    IF Error = 1 THEN 
        (* '<S2>:1:33' x = x0; *)
        PositionRef_m := fCylPos0_m;
        (* '<S2>:1:34' v = v0; *)
        VelocityRef_ms := fCylVel0_ms;
    ELSIF (fSimulationTime_s >= 0.0) AND (fSimulationTime_s < ft0_s) THEN 
        (* '<S2>:1:35' elseif t>=0 && t<t0 *)
        (* '<S2>:1:36' x = x0; *)
        PositionRef_m := fCylPos0_m;
        (* '<S2>:1:37' v = v0; *)
        VelocityRef_ms := fCylVel0_ms;
    ELSIF (fSimulationTime_s >= ft0_s) AND (fSimulationTime_s < x2_tmp_tmp) THEN 
        (* '<S2>:1:38' elseif t>=t0 && t<(t0+t1) *)
        (* '<S2>:1:39' x = x0 + v0*(t-t0)-(slopeExt/t1)*(t-t0)^2/2; *)
        slopeRetr := fSimulationTime_s - ft0_s;
        PositionRef_m := ((slopeRetr * fCylVel0_ms) + fCylPos0_m) - ((x1_tmp_tmp * (slopeRetr * slopeRetr)) / 2.0);
        (* '<S2>:1:40' v = v0-(slopeExt/t1)*(t-t0); *)
        VelocityRef_ms := fCylVel0_ms - (x1_tmp_tmp * slopeRetr);
    ELSIF (fSimulationTime_s >= x2_tmp_tmp) AND (fSimulationTime_s < x2_tmp) THEN 
        (* '<S2>:1:41' elseif t>=(t0+t1) && t<(t0+t1+t2) *)
        (* '<S2>:1:42' x = x1 + vs*(t-(t0+t1)); *)
        PositionRef_m := ((fSimulationTime_s - x2_tmp_tmp) * fVelocitySP_ms) + x1;
        (* '<S2>:1:43' v = vs; *)
        VelocityRef_ms := fVelocitySP_ms;
    ELSIF (fSimulationTime_s >= x2_tmp) AND (fSimulationTime_s < x4_tmp_tmp) THEN 
        (* '<S2>:1:44' elseif t>=(t0+t1+t2) && t<(t0+t1+t2+t3) *)
        (* '<S2>:1:45' x = x2+vs*(t-(t0+t1+t2))+(slopeExt/t3)*(t-(t0+t1+t2))^2/2; *)
        slopeRetr := fSimulationTime_s - ((ft0_s + ftRamp_s) + tHold);
        PositionRef_m := ((slopeRetr * fVelocitySP_ms) + x2) + ((x1_tmp_tmp * (slopeRetr * slopeRetr)) / 2.0);
        (* '<S2>:1:46' v = vs+(slopeExt/t3)*(t-(t0+t1+t2)); *)
        VelocityRef_ms := (slopeRetr * (slopeExt / ftRamp_s)) + fVelocitySP_ms;
    ELSIF (fSimulationTime_s >= x4_tmp_tmp) AND (fSimulationTime_s < x4_tmp) THEN 
        (* '<S2>:1:47' elseif t>=(t0+t1+t2+t3) && t<(t0+t1+t2+t3+t4) *)
        (* '<S2>:1:48' x = x_ref; *)
        PositionRef_m := fPositionSP_m;
        (* '<S2>:1:49' v = v0; *)
        VelocityRef_ms := fCylVel0_ms;
    ELSE 
        x1_tmp_tmp := ((x2_tmp_tmp + tHold) + ftRamp_s) + ftHoldPos_s;
        slopeExt := x1_tmp_tmp + ftRamp_s;

        IF (fSimulationTime_s >= x1_tmp_tmp) AND (fSimulationTime_s < slopeExt) THEN 
            (* '<S2>:1:50' elseif t>=(t0+t1+t2+t3+t4) && t<(t0+t1+t2+t3+t4+t5) *)
            (* '<S2>:1:51' x = x_ref - v0*(t-(t0+t1+t2+t3+t4))+(slopeRetr/t5)*(t-(t0+t1+t2+t3+t4))^2/2; *)
            tHold := fSimulationTime_s - x1_tmp_tmp;
            slopeRetr := slopeRetr / ftRamp_s;
            PositionRef_m := (fPositionSP_m - (tHold * fCylVel0_ms)) + ((slopeRetr * (tHold * tHold)) / 2.0);
            (* '<S2>:1:52' v = v0+(slopeRetr/t5)*(t-(t0+t1+t2+t3+t4)); *)
            VelocityRef_ms := (tHold * slopeRetr) + fCylVel0_ms;
        ELSE 
            x1_tmp_tmp := slopeExt + tHold;

            IF (fSimulationTime_s >= slopeExt) AND (fSimulationTime_s < x1_tmp_tmp) THEN 
                (* '<S2>:1:53' elseif t>=(t0+t1+t2+t3+t4+t5) && t<(t0+t1+t2+t3+t4+t5+t6) *)
                (* '<S2>:1:54' x = x4-vs*(t-(t0+t1+t2+t3+t4+t5)); *)
                PositionRef_m := x4 - ((fSimulationTime_s - slopeExt) * fVelocitySP_ms);
                (* '<S2>:1:55' v = -vs; *)
                VelocityRef_ms :=  -fVelocitySP_ms;
            ELSIF (fSimulationTime_s >= x1_tmp_tmp) AND (fSimulationTime_s < (x1_tmp_tmp + ftRamp_s)) THEN 
                (* '<S2>:1:56' elseif t>=(t0+t1+t2+t3+t4+t5+t6) && t<(t0+t1+t2+t3+t4+t5+t6+t7) *)
                (* '<S2>:1:57' x = x5-vs*(t-(t0+t1+t2+t3+t4+t5+t6))-(slopeRetr/t3)*(t-(t0+t1+t2+t3+t4+t5+t6))^2/2; *)
                tHold := fSimulationTime_s - x1_tmp_tmp;
                slopeRetr := slopeRetr / ftRamp_s;
                PositionRef_m := ((x4 - ((x1_tmp_tmp - slopeExt) * fVelocitySP_ms)) - (tHold * fVelocitySP_ms)) - ((slopeRetr * (tHold * tHold)) / 2.0);
                (* '<S2>:1:58' v = -vs-(slopeRetr/t3)*(t-(t0+t1+t2+t3+t4+t5+t6)); *)
                VelocityRef_ms := ( -fVelocitySP_ms) - (tHold * slopeRetr);
            ELSE 
                (* '<S2>:1:59' else *)
                (* '<S2>:1:60' x = x0; *)
                PositionRef_m := fCylPos0_m;
                (* '<S2>:1:61' v = v0; *)
                VelocityRef_ms := fCylVel0_ms;
            END_IF;

        END_IF;

    END_IF;

    (* '<S2>:1:63' T = t0+t1+t2+t3+t4+t5+t6+t7; *)
ELSE 
    (* '<S2>:1:64' else *)
    (* '<S2>:1:65' if Error == 1 *)

    IF Error = 1 THEN 
        (* '<S2>:1:66' x = x0; *)
        PositionRef_m := fCylPos0_m;
        (* '<S2>:1:67' v = v0; *)
        VelocityRef_ms := fCylVel0_ms;
    ELSIF (fSimulationTime_s >= 0.0) AND (fSimulationTime_s < ft0_s) THEN 
        (* '<S2>:1:68' elseif t>=0 && t<t0 *)
        (* '<S2>:1:69' x = x0; *)
        PositionRef_m := fCylPos0_m;
        (* '<S2>:1:70' v = v0; *)
        VelocityRef_ms := fCylVel0_ms;
    ELSIF (fSimulationTime_s >= ft0_s) AND (fSimulationTime_s < x2_tmp_tmp) THEN 
        (* '<S2>:1:71' elseif t>=t0 && t<(t0+t1) *)
        (* '<S2>:1:72' x = x0 + v0*(t-t0)-(slopeExt/t1)*(t-t0)^2/2; *)
        slopeRetr := fSimulationTime_s - ft0_s;
        PositionRef_m := (((fSimulationTime_s - ft0_s) * fCylVel0_ms) + fCylPos0_m) - ((x1_tmp_tmp * (slopeRetr * slopeRetr)) / 2.0);
        (* '<S2>:1:73' v = v0-(slopeExt/t1)*(t-t0); *)
        VelocityRef_ms := fCylVel0_ms - ((slopeExt / ftRamp_s) * slopeRetr);
    ELSIF (fSimulationTime_s >= x2_tmp_tmp) AND (fSimulationTime_s < x2_tmp) THEN 
        (* '<S2>:1:74' elseif t>=(t0+t1) && t<(t0+t1+t2) *)
        (* '<S2>:1:75' x = x1 + vs*(t-(t0+t1)); *)
        PositionRef_m := ((fSimulationTime_s - (ft0_s + ftRamp_s)) * fVelocitySP_ms) + x1;
        (* '<S2>:1:76' v = vs; *)
        VelocityRef_ms := fVelocitySP_ms;
    ELSIF (fSimulationTime_s >= x2_tmp) AND (fSimulationTime_s < x4_tmp_tmp) THEN 
        (* '<S2>:1:77' elseif t>=(t0+t1+t2) && t<(t0+t1+t2+t3) *)
        (* '<S2>:1:78' x = x2+vs*(t-(t0+t1+t2))+(slopeExt/t3)*(t-(t0+t1+t2))^2/2; *)
        slopeRetr := fSimulationTime_s - ((ft0_s + ftRamp_s) + tHold);
        slopeExt := slopeExt / ftRamp_s;
        PositionRef_m := ((slopeRetr * fVelocitySP_ms) + x2) + ((slopeExt * (slopeRetr * slopeRetr)) / 2.0);
        (* '<S2>:1:79' v = vs+(slopeExt/t3)*(t-(t0+t1+t2)); *)
        VelocityRef_ms := (slopeRetr * slopeExt) + fVelocitySP_ms;
    ELSE 
        (* '<S2>:1:80' else *)
        (* '<S2>:1:81' x = x_ref; *)
        PositionRef_m := fPositionSP_m;
        (* '<S2>:1:82' v = v0; *)
        VelocityRef_ms := fCylVel0_ms;
    END_IF;

    (* '<S2>:1:84' T = t0+t1+t2+t3+t4; *)
END_IF;

(* End of MATLAB Function: '<S1>/RampSignal' *)


(* Switch: '<S1>/Switch' incorporates:
 *  Switch: '<S1>/Switch1' *)

IF  NOT bEnable THEN 
    (* Outport: '<Root>/VelocityRef_ms' *)
    VelocityRef_ms := fCylVel0_ms;
    (* Outport: '<Root>/PositionRef_m' *)
    PositionRef_m := fCylPos0_m;
END_IF;

(* End of Switch: '<S1>/Switch' *)
(* End of Outputs for SubSystem: '<Root>/FB_RampMotionGenerator' *)

END_FUNCTION_BLOCK

// ---- StablePlatform/Function Blocks/FB_WaveMotionGenerator.TcPOU
FUNCTION_BLOCK FB_WaveMotionGenerator
VAR_INPUT
	bEnable: BOOL;
	fBias_deg: LREAL;
	fTheta0_deg: LREAL;
	fFreq_rads: LREAL;
	Fphase_rad: LREAL;
	fCyclicTime_s: LREAL;
END_VAR
VAR_OUTPUT
	fOmega_degs: LREAL;
	fTheta_deg: LREAL;
END_VAR
VAR
	fTheta_deg_tmp: LREAL;
END_VAR


(* Outputs for Atomic SubSystem: '<Root>/FB_WaveMotionGenerator' *)
(* Switch: '<S1>/Switch1' incorporates:
 *  Switch: '<S1>/Switch2' *)
(* y=amplitude×sin(frequency×time+phase)+bias *)
(* if t>=t0 && t<tFinal *)
(* x = x0+A*sin(w*(t-t0)); *)
(* xDot = w*A*cos(w*(t-t0)); *)
(* MATLAB Function 'FB_WaveMotionGenerator/WaveSignal': '<S2>:1' *)
(* '<S2>:1:6' x = A*cos(w*t+phase) + x0; *)
(* '<S2>:1:7' xDot = -w*A*sin(w*t+phase); *)
(* else  *)
(* x = x0;  *)
(* xDot = 0; *)
(* end *)

IF bEnable THEN 
    (* MATLAB Function: '<S1>/WaveSignal' *)
    fTheta_deg_tmp := (fFreq_rads * fCyclicTime_s) + Fphase_rad;
    (* Outport: '<Root>/fTheta_deg' incorporates:
     *  MATLAB Function: '<S1>/WaveSignal' *)
    fTheta_deg := (COS(fTheta_deg_tmp) * fTheta0_deg) + fBias_deg;
    (* Outport: '<Root>/fOmega_degs' incorporates:
     *  MATLAB Function: '<S1>/WaveSignal' *)
    fOmega_degs := SIN(fTheta_deg_tmp) * (( -fFreq_rads) * fTheta0_deg);
ELSE 
    (* Outport: '<Root>/fTheta_deg' *)
    fTheta_deg := fTheta0_deg;
    (* Outport: '<Root>/fOmega_degs' incorporates:
     *  Constant: '<S1>/Constant' *)
    fOmega_degs := 0.0;
END_IF;

(* End of Switch: '<S1>/Switch1' *)
(* End of Outputs for SubSystem: '<Root>/FB_WaveMotionGenerator' *)

END_FUNCTION_BLOCK

// ---- StablePlatform/Functions/F_PlatformAnglePos2CylPos.TcPOU
FUNCTION F_PlatformAnglePos2CylPos : LREAL
VAR_INPUT
	fPlatformAngleTheta1Ref : LREAL;
END_VAR
VAR
	pi : LREAL := 3.14159265;
	fMinLengthPlatformCylinder : LREAL := 0.878;
	fOffsetAngleDeg : LREAL := 55.4;
	fOffsetAngleRad : LREAL	:= fOffsetAngleDeg*pi/180;
	fLengthA : LREAL	:= 0.513; 
	fLengthC : LREAL	:= 1.353; 
	fAngleBeta : LREAL;
	fCylinderLength : LREAL; 
END_VAR

fAngleBeta := fPlatformAngleTheta1Ref - fOffsetAngleRad;

fCylinderLength := SQRT(fLengthA*fLengthA + fLengthC*fLengthC - 2*fLengthA*fLengthC*COS(fAngleBeta));

F_PlatformAnglePos2CylPos := fCylinderLength - fMinLengthPlatformCylinder;

END_FUNCTION

// ---- StablePlatform/Functions/F_deg2rad.TcPOU
FUNCTION F_deg2rad : LREAL
VAR_INPUT
	fInputRad : LREAL;
END_VAR
VAR
	pi : LREAL := 3.14159265;
END_VAR

F_deg2rad := (pi/180)*fInputRad;

END_FUNCTION

// ---- StablePlatform/Functions/F_PlatformAngleVel2CylVel.TcPOU
FUNCTION F_PlatformAngleVel2CylVel : LREAL
VAR_INPUT
	fPlatformAngleTheta1Ref : LREAL;
	fPlatformAngleOmega1Ref : LREAL;
END_VAR
VAR
	pi : LREAL := 3.14159265;
	fMinLengthPlatformCylinder : LREAL := 0.878;
	fOffsetAngleDeg : LREAL := 55.4;
	fOffsetAngleRad : LREAL	:= fOffsetAngleDeg*pi/180;
	fLengthA : LREAL	:= 0.513; 
	fLengthC : LREAL	:= 1.353; 
	fAngleBeta : LREAL;
	fCylinderLength : LREAL; 
	K : LREAL;
END_VAR

fAngleBeta := fPlatformAngleTheta1Ref - fOffsetAngleRad;

fCylinderLength := SQRT(fLengthA*fLengthA + fLengthC*fLengthC - 2*fLengthA*fLengthC*COS(fAngleBeta));

K := fLengthA*fLengthA + fLengthC*fLengthC - 2 * fLengthA * fLengthC * COS(fAngleBeta);

F_PlatformAngleVel2CylVel := (fLengthA * fLengthC * SIN(fAngleBeta)) / SQRT(K)*fPlatformAngleOmega1Ref;

END_FUNCTION

// ---- StablePlatform/Function Blocks/FB_LowpassFilter.TcPOU
FUNCTION_BLOCK FB_LowpassFilter
VAR_INPUT
	fInput 				: LREAL;		      // Input
	fDeltaT				: LREAL; 			 // Cycle time [s]
	// Tuning Parameters 
	fCutoffFreq 		: LREAL := 0.5; 	  // seconds, value of 0 disables the filter
	fDamping 			: LREAL := 1/SQRT(2); // Damping ratio --> 0.707106781186547
	// Optional Parameters (Dont need to be used)
	bEnableLimits		: BOOL := FALSE;
	fLimitMax			: LREAL := 1.0;
	fLimitMin 			: LREAL := -1.0;
	// Optional Inputs (Dont need to be used)
	fDotInput_bypass 	: LREAL := 0;	      // Additional velocity input that bypasses the filter [unit/s]
	bReset 				: BOOL;				 // Resets the filter, and Sets Output = Input
END_VAR
VAR_OUTPUT
	fOutput 			: LREAL := fInput;	 // Output
	bError 				: BOOL;				 // TRUE if error
END_VAR
VAR
	fC 				: LREAL;
	fC2 			: LREAL; // c^2
	fDotOuptut 	: LREAL;
	fDot2Ouptut 	: LREAL;
	bFirstRun 		: BOOL := TRUE;
END_VAR

bError := FALSE;

IF (fCutoffFreq < 1E-10) THEN
	fOutput := fInput;
	bReset := TRUE;
END_IF

IF NOT bReset THEN
	fC := 2*PI*fDeltaT/fCutoffFreq;
	IF (fC <= 0) THEN
		bError := TRUE;
		bReset := TRUE;
	ELSIF (fC >= 0.9) THEN
		fC := 0.9;
	END_IF
END_IF

IF bReset OR bFirstRun THEN
	bFirstRun := FALSE;
	bReset := FALSE;
	fOutput := fInput;
	fDotOuptut  := 0;
	fDot2Ouptut := 0;
	RETURN;
END_IF

IF bError THEN RETURN; END_IF

fC2 := EXPT(fC, 2.0);

fDot2Ouptut := (fInput - fOutput)*fC2 - 2*fDamping*fC*fDotOuptut;

fDotOuptut := fDotOuptut + fDot2Ouptut;
fOutput := fOutput + fDotOuptut + fDotInput_bypass*fDeltaT;

IF ABS(fOutput) < 1E-10 THEN
	fOutput := 0;
END_IF

IF bEnableLimits THEN
	fOutput := LIMIT(fLimitMin,fOutput,fLimitMax);	
ELSE 
	fOutput := fOutput; 
END_IF

END_FUNCTION_BLOCK

// ---- StablePlatform/Functions/F_rad2deg.TcPOU
FUNCTION F_rad2deg : LREAL
VAR_INPUT
	fInputDeg : LREAL;
END_VAR
VAR
	pi : LREAL := 3.14159265;
END_VAR

F_rad2deg := (180/pi)*fInputDeg;

END_FUNCTION

// ---- StablePlatform/Functions/fPlatformAngleTheta1.TcPOU
FUNCTION fPlatformAngleTheta1 : LREAL
VAR_INPUT
	fStroke : LREAL;
END_VAR
VAR
	fAngleBeta		: LREAL;
	fCylinderLength	: LREAL;
	fMinLength 		: LREAL; 
END_VAR

fMinLength := G_StablePlatformParameters.fMinLengthPlatformCylinder;

fCylinderLength := fStroke + fMinLength;

fAngleBeta := ACOS((G_StablePlatformParameters.fLengthA*G_StablePlatformParameters.fLengthA +  G_StablePlatformParameters.fLengthC*G_StablePlatformParameters.fLengthC - fCylinderLength*fCylinderLength) / (2 * G_StablePlatformParameters.fLengthA * G_StablePlatformParameters.fLengthC));

fPlatformAngleTheta1 := -(fAngleBeta - G_StablePlatformParameters.fOffsetAngleRad);

END_FUNCTION

// ---- StablePlatform/Function Blocks/FB_AnalogInputScalingPlusMinus.TcPOU
FUNCTION_BLOCK FB_AnalogInputScalingPlusMinus
VAR_INPUT
	nRawInput 				: INT;
	stAnalogInputScaling    : ST_AnalogInputScaling_1;
END_VAR
VAR_OUTPUT
	fOutput 				: LREAL;
END_VAR
VAR
	fRawInput 				: LREAL;
	fNormalizedInput		: LREAL;
END_VAR

fRawInput := INT_TO_LREAL(nRawInput);

fNormalizedInput := (stAnalogInputScaling.fMaxOutputValue - stAnalogInputScaling.fMinOutputValue)/2 + (fRawInput/stAnalogInputScaling.fMaxInputValue)*((stAnalogInputScaling.fMaxOutputValue - stAnalogInputScaling.fMinOutputValue)/2);

fOutput := LIMIT(stAnalogInputScaling.fMinOutputValue, fNormalizedInput, stAnalogInputScaling.fMaxOutputValue);

//fNormalizedInput := (fRawInput - stAnalogInputScaling.fMinInputValue) / (stAnalogInputScaling.fMaxInputValue - stAnalogInputScaling.fMinInputValue);

//fOutput := LIMIT(stAnalogInputScaling.fMinOutputValue, stAnalogInputScaling.fMinOutputValue + fNormalizedInput*(stAnalogInputScaling.fMaxOutputValue - stAnalogInputScaling.fMinOutputValue), stAnalogInputScaling.fMaxOutputValue);

END_FUNCTION_BLOCK

// ---- StablePlatform/Function Blocks/FB_WaveMotionGenerator_1.TcPOU
FUNCTION_BLOCK FB_WaveMotionGenerator_1
VAR_INPUT
	bEnable: BOOL;
	fBias_deg: LREAL;
	fTheta0_deg: LREAL;
	fFreq_rads: LREAL;
	Fphase_rad: LREAL;
	fCyclicTime_s: LREAL;
END_VAR
VAR_OUTPUT
	fOmega_degs: LREAL;
	fTheta_deg: LREAL;
END_VAR
VAR
	fTheta_deg_tmp: LREAL;
END_VAR


(* Outputs for Atomic SubSystem: '<Root>/FB_WaveMotionGenerator' *)
(* Switch: '<S1>/Switch1' incorporates:
 *  Switch: '<S1>/Switch2' *)
(* y=amplitude×sin(frequency×time+phase)+bias *)
(* if t>=t0 && t<tFinal *)
(* x = x0+A*sin(w*(t-t0)); *)
(* xDot = w*A*cos(w*(t-t0)); *)
(* MATLAB Function 'FB_WaveMotionGenerator/WaveSignal': '<S2>:1' *)
(* '<S2>:1:6' x = A*cos(w*t+phase) + x0; *)
(* '<S2>:1:7' xDot = -w*A*sin(w*t+phase); *)
(* else  *)
(* x = x0;  *)
(* xDot = 0; *)
(* end *)

IF bEnable THEN 
    (* MATLAB Function: '<S1>/WaveSignal' *)
    fTheta_deg_tmp := (fFreq_rads * fCyclicTime_s) + Fphase_rad;
    (* Outport: '<Root>/fTheta_deg' incorporates:
     *  MATLAB Function: '<S1>/WaveSignal' *)
    fTheta_deg := (COS(fTheta_deg_tmp) * fTheta0_deg) + fBias_deg;
    (* Outport: '<Root>/fOmega_degs' incorporates:
     *  MATLAB Function: '<S1>/WaveSignal' *)
    fOmega_degs := SIN(fTheta_deg_tmp) * (( -fFreq_rads) * fTheta0_deg);
ELSE 
    (* Outport: '<Root>/fTheta_deg' *)
    fTheta_deg := fTheta0_deg;
    (* Outport: '<Root>/fOmega_degs' incorporates:
     *  Constant: '<S1>/Constant' *)
    fOmega_degs := 0.0;
END_IF;

(* End of Switch: '<S1>/Switch1' *)
(* End of Outputs for SubSystem: '<Root>/FB_WaveMotionGenerator' *)

END_FUNCTION_BLOCK

// ---- GlobalTextList.TcGTLO
TEXTLIST GlobalTextList
  136 = ' MaxPosError: %0.1f [mm]'
  879 = ' MaxValveFlow: %0.1f [l/min]'
  663 = '%0.1f  Amplitude (theta0 [deg])'
  49 = '%0.1f Amplitude (theta0 [deg])'
  845 = '%0.1f CylPos [m]'
  821 = '%0.1f CylPosRef [m]'
  261 = '%0.1f CylVel [m]'
  364 = '%0.1f CylVelRef [m/s]'
  891 = '%0.1f CylVelSp [m/s]'
  808 = '%0.1f CyVel0 [m/s]'
  93 = '%0.1f Freq [rad/s]'
  46 = '%0.1f MaxPosError [mm]'
  635 = '%0.1f MaxValveFlow [l/min]'
  762 = '%0.1f Pgain [-]'
  670 = '%0.1f PlatformPos [deg]'
  387 = '%0.1f PlatformPos0 [deg]'
  505 = '%0.1f PlatformPosRef [deg]'
  135 = '%0.1f PlatformPosSp [deg]'
  979 = '%0.1f PlatformVelRef [deg/s]'
  395 = '%0.1f t0 [s]'
  202 = '%0.1f tHold'
  696 = '%0.1f Time[s]'
  636 = '%0.1f tRamp [s]'
  24 = '%f'
  608 = '%f Amplitude (theta0 [deg])'
  695 = '%f Cylinder Position [m]'
  963 = '%f Cylinder Velocity [m/s]'
  487 = '%f CylPos [m]'
  344 = '%f CylPosRef [m]'
  503 = '%f CylVelRef [m/s]'
  284 = '%f CylVelSp [m/s]'
  40 = '%f CyVel0 [m/s]'
  887 = '%f Freq [rad/s]'
  620 = '%f Igain [-]'
  588 = '%f MaxPosError [mm]'
  767 = '%f MaxValveFlow [l/min]'
  253 = '%f Pgain [-]'
  766 = '%f PlatformPos [deg]'
  233 = '%f PlatformPos0 [deg]'
  175 = '%f PlatformPosRef [deg]'
  129 = '%f PlatformPosSp [deg]'
  568 = '%f PlatformVelRef [deg/s]'
  931 = '%f t0 [s]'
  468 = '%f tHold'
  332 = '%f Time[s]'
  431 = '%f tRamp [s]'
  47 = '%f [m]'
  798 = '24VDC PowerRefresh'
  519 = 'AcknowAledge'
  820 = 'Acknowledge'
  15 = 'Activated'
  23 = 'Active'
  201 = 'Amplitude: %0.1f  (theta0 [deg])'
  606 = 'Auto               Manual'
  985 = 'AutoModeControl'
  716 = 'CylPos: %f [m]'
  162 = 'CylPosRef  %f [m]'
  33 = 'CylPosRef: %f [m]'
  612 = 'CylVel: %f [m]'
  82 = 'CylVelRef: %f [m/s]'
  235 = 'CylVelSp: %f [m/s]'
  890 = 'Drive STO'
  810 = 'EMG Stop'
  418 = 'Enable'
  854 = 'Enable Full Periode'
  497 = 'Freq: %0.1f [rad/s]'
  942 = 'Group'
  463 = 'Group                                   Run/Stop'
  914 = 'Group Run/Stop'
  708 = 'GroupBox'
  25 = 'Igain: %0.1f [-]'
  990 = 'Integral Control'
  691 = 'MaxControlSignal: %0.1f [-]'
  248 = 'Mode'
  65 = 'Motion Controller'
  641 = 'Pgain: %0.1f [-]'
  908 = 'PlatformPos: %f [deg]'
  177 = 'PlatformPosRef: %f [deg]'
  698 = 'PlatformVelRef: %f [deg/s]'
  980 = 'Position Feedback Control'
  107 = 'PowerRefresh'
  27 = 'RampMotion'
  181 = 'Restart'
  267 = 'Run/Stop'
  114 = 'Stable Platform'
  246 = 'Start Motion'
  313 = 'Time: %0.1f [s]'
  488 = 'TwinSAFE'
  504 = 'Velocity Feed Forward'
  277 = 'Wave             Ramp'
  142 = 'WaveMotion'
END_TEXTLIST

// ---- HMI/HMI.TcVIS
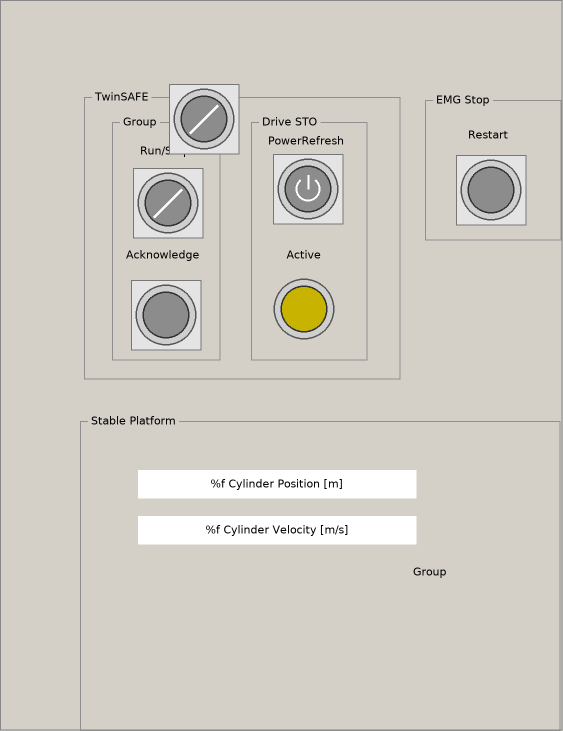
VISUALIZATION HMI  // 563x731
    GroupBox (84,89 316x290), "TwinSAFE"
        Label (268,468 156x30), "Group"
        Label (3,47 156x30), "Run/Stop"
        Label (1,151 156x30), "Acknowledge"
        GroupBox (28,25 108x246), "Group"
            RotarySwitch (21,54 70x70), variable: G_Safety_AXIS4.TwinSafeGroupRunStop, behaviour: TOGGLE, style: Switch-RotarySwitch-Gray
            PushSwitch (19,166 70x70), variable: G_Safety_AXIS4.TwinSafeGroupComErrAck, behaviour: TAP, style: Switch-PushSwitch-Gray
        Lamp1 (170,918 70x70), variable: G_Safety_AXIS4.ChA_STO_Active, style: Lamp-Lamp1-Yellow
        GroupBox (167,25 116x246), "Drive STO"
            RotarySwitch (-82,-30 70x70), behaviour: TOGGLE, style: Switch-RotarySwitch-Gray
            Lamp1 (18,160 70x70), variable: G_Safety_AXIS4.ChA_STO_Active, style: Lamp-Lamp1-Yellow
            PowerSwitch (22,40 70x70), variable: G_Safety_AXIS4.bWinchMotor24vDisable, behaviour: TAP, style: Switch-PowerSwitch-Gray
        Label (145,151 150x30), "Active"
        Label (147,37 150x30), "PowerRefresh"
    GroupBox (80,413 480x318), "Stable Platform"
        Textfield (57,56 280x30), "%f Cylinder Position [m]", text variable: G_StablePlatformScaledIO.fPistonPosition
        Textfield (57,102 280x30), "%f Cylinder Velocity [m/s]", text variable: G_StablePlatformScaledIO.fPistonVelocity
    GroupBox (425,92 136x148), "EMG Stop"
        PushSwitch (31,63 70x70), variable: G_Safety_AXIS4.EMGRestart, behaviour: TAP, style: Switch-PushSwitch-Gray
    Label (413,120 150x30), "Restart"
END_VISUALIZATION

// ---- StablePlatform/StablePlatform.TcVIS
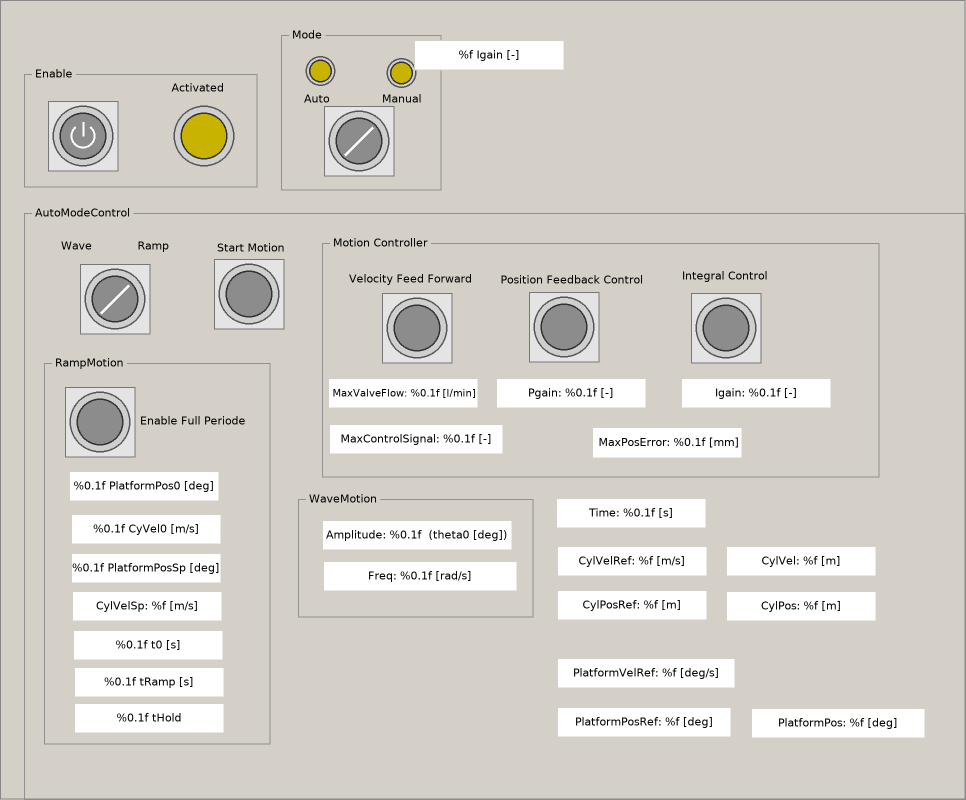
VISUALIZATION StablePlatform  // 966x800
    GroupBox (281,27 160x163), "Mode"
        RotarySwitch (43,79 70x70), variable: G_StablePlatformIO.bModeSelector, behaviour: TOGGLE, style: Switch-RotarySwitch-Gray
        Lamp1 (21,27 37x34), variable: G_StablePlatformIO.bAutoMode, style: Lamp-Lamp1-Yellow
        Lamp1 (102,29 37x34), variable: G_StablePlatformIO.bManualMode, style: Lamp-Lamp1-Yellow
        Label (7,57 150x30), "Auto Manual"
    GroupBox (24,66 233x121), "Enable"
        PowerSwitch (24,35 70x70), variable: G_StablePlatformIO.bEnable, behaviour: TOGGLE, style: Switch-PowerSwitch-Gray
        Lamp1 (145,35 70x70), variable: G_StablePlatformIO.bActivated, style: Lamp-Lamp1-Yellow
    GroupBox (24,205 942x595), "AutoModeControl"
        RotarySwitch (56,59 70x70), variable: G_StablePlatformIO.bMotionModeSelector, behaviour: TOGGLE, style: Switch-RotarySwitch-Gray
        Label (16,26 150x30), "Wave Ramp"
        PushSwitch (190,54 70x70), variable: G_StablePlatformIO.bStartMotionGenerator, behaviour: TOGGLE, style: Switch-PushSwitch-Gray
        Label (152,28 150x30), "Start Motion"
        GroupBox (20,150 226x389), "RampMotion"
            PushSwitch (21,32 70x70), variable: G_StablePlatformIO.bRampMotionFullPeriode, behaviour: TOGGLE, style: Switch-PushSwitch-Gray
            Label (74,51 150x30), "Enable Full Periode"
            Textfield (25,116 150x30), "%0.1f PlatformPos0 [deg]", text variable: G_StablePlatformIO.bRampMotionPos0_deg
                OnMouseDown: write the text variable via Default
            Textfield (27,159 150x30), "%0.1f CyVel0 [m/s]", text variable: G_StablePlatformIO.bRampMotionCylVel0_ms
                OnMouseDown: write the text variable via Default
            Textfield (27,198 150x30), "%0.1f PlatformPosSp [deg]", text variable: G_StablePlatformIO.bRampMotionPositionSP_deg
                OnMouseDown: write the text variable via Default
            Textfield (28,236 150x30), "CylVelSp: %f [m/s]", text variable: G_StablePlatformIO.bRampMotionVelocitySP_ms
                OnMouseDown: write the text variable via Default
            Textfield (29,275 150x30), "%0.1f t0 [s]", text variable: G_StablePlatformIO.bRampMotiont0_s
                OnMouseDown: write the text variable via Default
            Textfield (30,312 150x30), "%0.1f tRamp [s]", text variable: G_StablePlatformIO.bRampMotiontRamp_s
                OnMouseDown: write the text variable via Default
            Textfield (30,348 150x30), "%0.1f tHold", text variable: G_StablePlatformIO.bRampMotiontHoldPos_s
                OnMouseDown: write the text variable via Default
        Textfield (532,293 150x30), "Time: %0.1f [s]", text variable: G_StablePlatformIO.fTime
        GroupBox (274,286 235x126), "WaveMotion"
            Textfield (24,29 190x30), "Amplitude: %0.1f (theta0 [deg])", text variable: G_StablePlatformIO.fWaveMotionAplitudeTheta0_deg
                OnMouseDown: write the text variable via Default
            Textfield (25,70 194x30), "Freq: %0.1f [rad/s]", text variable: G_StablePlatformIO.WaveMotionFreq_rads
                OnMouseDown: write the text variable via Default
        Textfield (533,341 150x30), "CylVelRef: %f [m/s]", text variable: G_StablePlatformIO.fCylVelRef_ms
        Textfield (533,385 150x30), "CylPosRef: %f [m]", text variable: G_StablePlatformIO.fCylPosRef_m
        Textfield (702,386 150x30), "CylPos: %f [m]", text variable: G_StablePlatformScaledIO.fPistonPosition
        Textfield (702,341 150x30), "CylVel: %f [m]", text variable: G_StablePlatformScaledIO.fPistonVelocity
        Textfield (533,453 178x30), "PlatformVelRef: %f [deg/s]", text variable: G_StablePlatformIO.fWaveMotionOmega_degs
        Textfield (533,502 174x30), "PlatformPosRef: %f [deg]", text variable: G_StablePlatformIO.fWaveMotionTheta_deg
        Textfield (727,503 174x30), "PlatformPos: %f [deg]", text variable: G_StablePlatformScaledIO.fPlatformAngleDeg
        Textfield (390,-165 150x30), "%f Igain [-]", text variable: G_StablePlatformIO.fIntegralGain
        GroupBox (298,30 557x242), "Motion Controller"
            PushSwitch (60,58 70x70), variable: G_StablePlatformIO.bEnableFeedForward, behaviour: TOGGLE, style: Switch-PushSwitch-Gray
            PushSwitch (207,57 70x70), variable: G_StablePlatformIO.bEnableFeedBackControl, behaviour: TOGGLE, style: Switch-PushSwitch-Gray
            PushSwitch (369,58 70x70), variable: G_StablePlatformIO.bEnableIntegralControl, behaviour: TOGGLE, style: Switch-PushSwitch-Gray
            Textfield (270,192 150x31), "MaxPosError: %0.1f [mm]", text variable: G_StablePlatformIO.fMaxPosError_mm
                OnMouseClick: write the text variable via Default
            Textfield (174,143 150x30), "Pgain: %0.1f [-]", text variable: G_StablePlatformIO.fProportionalGain
                OnMouseClick: write the text variable via Default, min 0.0000001
            Textfield (6,143 150x30), "MaxValveFlow: %0.1f [l/min]", text variable: G_StablePlatformIO.fMaxValveFlow_lmin
                OnMouseClick: write the text variable via Default
            Textfield (359,143 150x30), "Igain: %0.1f [-]", text variable: G_StablePlatformIO.fIntegralGain
                OnMouseClick: write the text variable via Default
            Label (175,30 150x30), "Position Feedback Control"
            Label (328,26 150x30), "Integral Control"
            Textfield (7,189 174x30), "MaxControlSignal: %0.1f [-]", text variable: G_StablePlatformParameters.fMaxControlSignal
                OnMouseClick: write the text variable via Default, min -1, max 1
        Label (297,59 179x30), "Velocity Feed Forward"
    Label (123,73 150x30), "Activated"
END_VISUALIZATION
